// TIA Portal V20 export
TYPE "LKinCtrl_typeMovePickAndPlaceParameters"
   STRUCT
      startParameter : "LKinCtrl_typePnPParameter";   // Start vector parameter
      targetParameter : "LKinCtrl_typePnPParameter";   // Target vector parameter
   END_STRUCT;
END_TYPE
